FUNCTION_BLOCK PedCrossingCtl (* Basic Function Block Type *)
  (* Standard: 61499-2 *)
  (* Version 0.0, 2014-07-14, 4DIAC-IDE, 4DIAC-Consortium *)
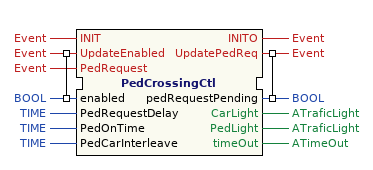
  EVENT_INPUT
    INIT; (* Initialization Request *)
    UpdateEnabled WITH enabled;
    PedRequest;
  END_EVENT
  EVENT_OUTPUT
    INITO;
    UpdatePedReq WITH pedRequestPending;
  END_EVENT
  VAR_INPUT
    enabled : BOOL; (* determines if this crossing is enabled, if currently the pedestrian walk is green the pedestrian cycle will be finished before a full disable of the crossing is performed *)
    PedRequestDelay : TIME;
    PedOnTime : TIME;
    PedCarInterleave : TIME;
  END_VAR
  VAR_OUTPUT
    pedRequestPending : BOOL;
  END_VAR
  PLUGS
    CarLight : ATraficLight;
    PedLight : ATraficLight;
    timeOut : ATimeOut;
  END_PLUGS
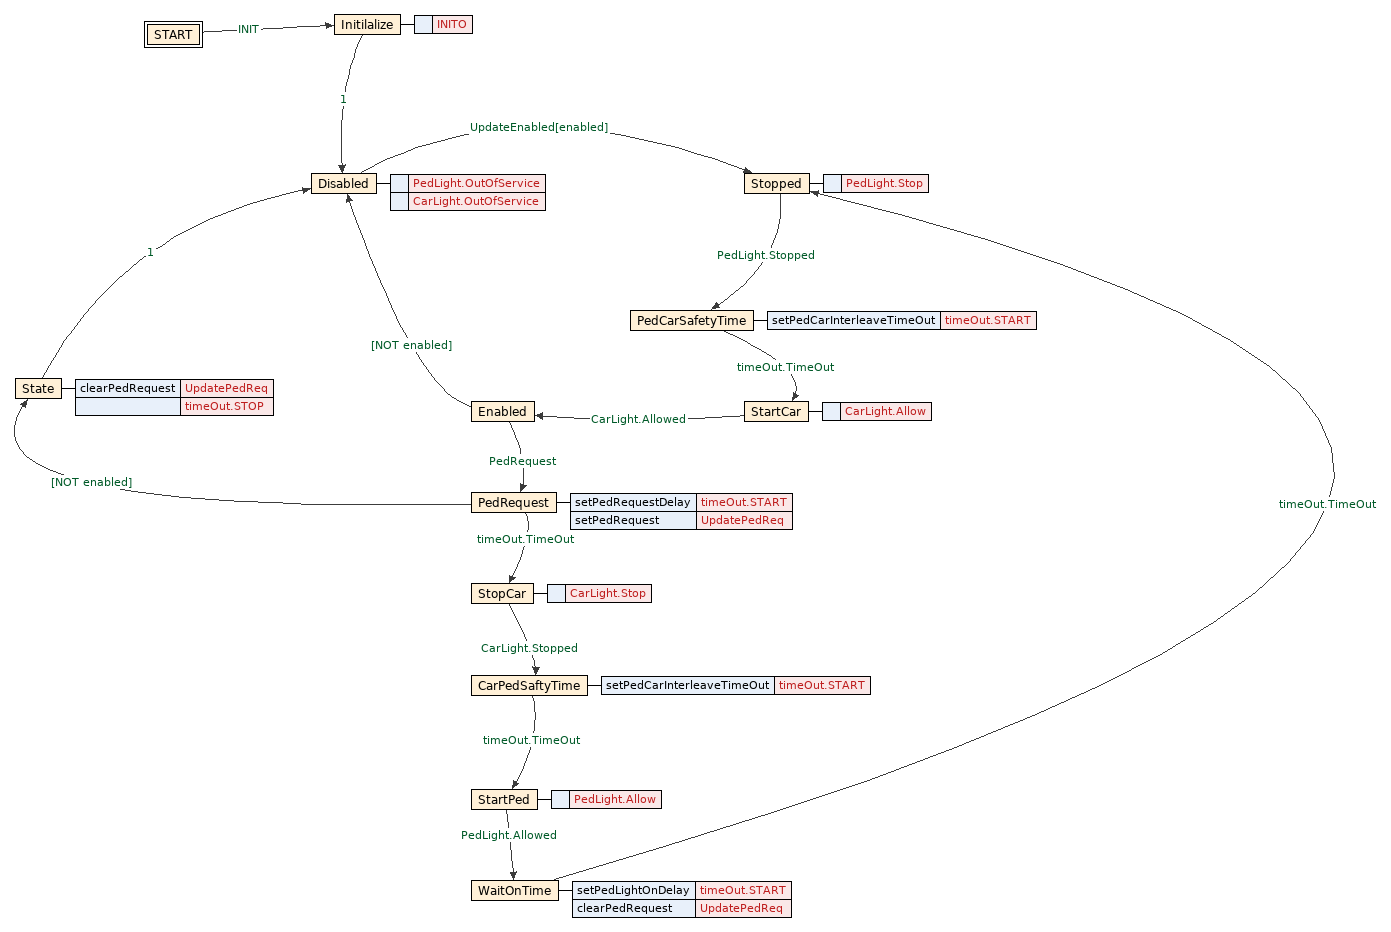
  EC_STATES
    START; (* Initial State *)
    Disabled : -> PedLight.OutOfService, -> CarLight.OutOfService; (* Initialization *)
    Stopped : -> PedLight.Stop;
    StartCar : -> CarLight.Allow;
    Enabled;
    PedRequest : setPedRequestDelay -> timeOut.START, setPedRequest -> UpdatePedReq;
    StopCar : -> CarLight.Stop;
    StartPed : -> PedLight.Allow;
    WaitOnTime : setPedLightOnDelay -> timeOut.START, clearPedRequest -> UpdatePedReq;
    CarPedSaftyTime : setPedCarInterleaveTimeOut -> timeOut.START;
    PedCarSafetyTime : setPedCarInterleaveTimeOut -> timeOut.START;
    Initilalize : -> INITO;
    State : clearPedRequest -> UpdatePedReq, -> timeOut.STOP;
  END_STATES
  EC_TRANSITIONS
    Disabled TO Stopped := UpdateEnabled[enabled];
    StartCar TO Enabled := CarLight.Allowed;
    Enabled TO Disabled := [NOT enabled];
    Enabled TO PedRequest := PedRequest;
    PedRequest TO StopCar := timeOut.TimeOut;
    StartPed TO WaitOnTime := PedLight.Allowed;
    WaitOnTime TO Stopped := timeOut.TimeOut;
    StopCar TO CarPedSaftyTime := CarLight.Stopped;
    CarPedSaftyTime TO StartPed := timeOut.TimeOut;
    Stopped TO PedCarSafetyTime := PedLight.Stopped;
    PedCarSafetyTime TO StartCar := timeOut.TimeOut;
    START TO Initilalize := INIT;
    Initilalize TO Disabled := 1;
    PedRequest TO State := [NOT enabled];
    State TO Disabled := 1;
  END_TRANSITIONS
  ALGORITHM setPedRequestDelay IN ST: (* Initialization algorithm *)
timeOut.DT := PedRequestDelay;
  END_ALGORITHM
  ALGORITHM setPedLightOnDelay IN ST: (* Normally executed algorithm *)
timeOut.DT := PedOnTime;
  END_ALGORITHM
  ALGORITHM setPedCarInterleaveTimeOut IN ST:
timeOut.DT := PedCarInterleave;
  END_ALGORITHM
  ALGORITHM setPedRequest IN ST: (* set the ped Requst pending bit to true *)
pedRequestPending := TRUE;
  END_ALGORITHM
  ALGORITHM clearPedRequest IN ST: (* new algorithm *)
pedRequestPending := FALSE;
  END_ALGORITHM
END_FUNCTION_BLOCK
